// TwinCAT 3 PLC project MasterArmControl
// ProgramVersion: 3.1.4024.0
// libraries:
//   Tc2_Math, * (Beckhoff Automation GmbH)
//   Tc2_Standard, * (Beckhoff Automation GmbH)
//   Tc2_System, * (Beckhoff Automation GmbH)
//   Tc3_Module, * (Beckhoff Automation GmbH)
// project tree:
//   Controllers/ FB_ADD.TcPOU, FB_Test.TcPOU, ITF.TcIO
//   DUTs/Enum/ E_DriverCtrlWord.TcDUT, E_DriverOPMode.TcDUT (not stored), E_DriverStatusWord.TcDUT (not stored), E_InstrumentType.TcDUT, E_MasterArmState.TcDUT, E_MatchedSlaveArmIdx.TcDUT, E_SlaveArmState.TcDUT
//   DUTs/Structure/ ST_CartStatus.TcDUT, ST_Frame.TcDUT (not stored), ST_InstruStatus.TcDUT (not stored), ST_MasterStatus.TcDUT, ST_MotorInputs.TcDUT, ST_MotorOutputs.TcDUT (not stored), ST_SlaveStatus.TcDUT (not stored)
//   DUTs/Type/ Mat3d.TcDUT (not stored), Vec3d.TcDUT (not stored), Vec6d.TcDUT (not stored), Vec7d.TcDUT (not stored), Vec7i.TcDUT (not stored)
//   FBs_Controller/ FB_MasterArmCtrlBase.TcPOU, FB_PID.TcPOU (not stored), FBRedunOriControl.TcPOU, I_MasterArmCtrl.TcIO
//   FBs_dynamics/ FB_MasterGravity.TcPOU, FB_MasterGravity_1.TcPOU (not stored)
//   FBs_Filter/ FB_LowPassFilter.TcPOU (not stored)
//   GVLs/ GVL_ArmParameters.TcGVL, GVL_CartParameters.TcGVL, GVL_ControlParameters.TcGVL, GVL_MathDefine.TcGVL, GVL_MotorParameters.TcGVL (not stored), GVL_SafetyParameters.TcGVL (not stored), GVL_SystemParameters.TcGVL (not stored)
//   / MAIN.TcPOU, PlcTask.TcTTO (not stored)
//   Maths/ addVec3.TcPOU, atan2.TcPOU (not stored), cot.TcPOU, mat3Mat3.TcPOU (not stored), mat3Vec3.TcPOU, mat67Vec7.TcPOU, rotZ.TcPOU, rotY.TcPOU (not stored), rotX.TcPOU, transform.TcPOU
//   Robots/ FB_Joint.TcPOU, FB_MasterArm.TcPOU, FB_MasterRobot.TcPOU
// real-time tasks:
//   TASK PlcTask: cycle T#10ms, priority 20, ADS port 350

// ---- DUTs/Enum/E_DriverCtrlWord.TcDUT
TYPE E_DriverCtrlWord :
(
	DriverCtrlWord_INIT := 6,
	DriverCtrlWord_PREOP := 7,
	DriverCtrlWord_OP := 15
);
END_TYPE

// ---- DUTs/Enum/E_InstrumentType.TcDUT
TYPE E_InstrumentType :
(
	InstruType_UNKNOWM := 0,
	InstruType_endoscope := 1,
	InstruType_NeedleGripper := 2,
	InstruType_Energy :=3
);
END_TYPE

// ---- DUTs/Enum/E_MasterArmState.TcDUT
TYPE E_MasterArmState :
(
	MasterArmState_Errot := 0,
	MasterArmState_Cart := 1,
	MasterArmState_Init :=2,
	MasterArmState_Home :=3,
	MasterArmState_Standby :=4,
	MasterArmState_Matching :=5,
	MasterArmState_Ready :=6,
	MasterArmState_MasterSlave :=7,
	MasterArmState_Clutch :=8,
	MasterArmState_Endoscope :=9
);
END_TYPE

// ---- DUTs/Enum/E_MatchedSlaveArmIdx.TcDUT
TYPE E_MatchedSlaveArmIdx :
(
	MatchedSlaveArmIdx_NULL := 0,
	MatchedSlaveArmIdx_1 := 1,
	MatchedSlaveArmIdx_2 := 2,
	MatchedSlaveArmIdx_3 := 3,
	MatchedSlaveArmIdx_4 := 4
);
END_TYPE

// ---- DUTs/Enum/E_SlaveArmState.TcDUT
TYPE E_SlaveArmState :
(
	SlaveArmState_Errot := 0,
	SlaveArmState_Cart := 1,
	SlaveArmState_Init :=2,
	SlaveArmState_Standby :=3,
	SlaveArmState_InstallPanel:=4,
	SlaveArmState_PanelReady :=5,
	SlaveArmState_InstallInstru :=6,
	SlaveArmState_InstruReady :=7,
	SlaveArmState_MasterSlave :=8,
	SlaveArmState_InstallScope :=9,
	SlaveArmState_ScopeReady :=10,
	SlaveArmState_EndoScope :=11
);
END_TYPE

// ---- DUTs/Structure/ST_CartStatus.TcDUT
TYPE ST_CartStatus :
STRUCT
	m_monitorAngle:LREAL := 0.0;
	m_armSwitch:BOOL := FALSE;
	m_clutchSwitch:BOOL := FALSE;
	m_endoscopeSwitch:BOOL := FALSE;
	m_instrumentPowerSwitch:BOOL := FALSE;
	m_monitorAdjustSwitch:BOOL := FALSE;
	m_tableAdjustSwitch:BOOL := FALSE;
END_STRUCT
END_TYPE

// ---- DUTs/Structure/ST_MasterStatus.TcDUT
TYPE ST_MasterStatus :
STRUCT
	// state machine
	m_armState:ARRAY[1..g_mArmNum] OF E_masterArmState;
	
	// index(0 to 4) of slave arm which is tele-linked to master arm
	m_slaveArmIdx :ARRAY[1..g_mArmNum] OF INT;
	
	// grip angle
	m_gripAngle:ARRAY[1..g_mArmNum] OF LREAL;
	
	// command arm pose in monitor
	m_cmdArmPose :ARRAY[1..g_mArmNum] OF ST_Frame;
	
	// current arm pose in monitor
	m_curArmPose:ARRAY[1..g_mArmNum] OF ST_Frame;
	
	// command arm twist[linear velocity; angular veloicty] in monitor
	m_cmdArmTwist:ARRAY[1..g_mArmNum,1..6] OF LREAL;
	
	// current arm twist[linear velocity; angular veloicty] in monitor
	m_curArmTwist:ARRAY[1..g_mArmNum,1..6] OF LREAL;
	
	// joint position compute with motor encoder
	m_curMotorPos :ARRAY[1..g_mJntNum] OF LREAL;
	
	// joint position compute with link/abs encoder
	m_curLinkPos :ARRAY[1..g_mArmNum, 1..g_mJntNum] OF LREAL;
	
	// target joint position 
	m_cmdJntPos :ARRAY[1..g_mArmNum, 1..g_mJntNum] OF LREAL;
	
	// current joint position 
	m_curJntPos :ARRAY[1..g_mArmNum, 1..g_mJntNum] OF LREAL;
	
	// target joint velocity 
	m_cmdJntVel :ARRAY[1..g_mArmNum, 1..g_mJntNum] OF LREAL;
	
	// current joint position 
	m_curJntVel :ARRAY[1..g_mArmNum, 1..g_mJntNum] OF LREAL;
	
	// command joint torque 
	m_cmdJntTrq :ARRAY[1..g_mArmNum, 1..g_mJntNum] OF LREAL;
	
	// current joint torque 
	m_curJntTrq :ARRAY[1..g_mArmNum, 1..g_mJntNum] OF LREAL;
	
END_STRUCT
END_TYPE

// ---- DUTs/Structure/ST_MotorInputs.TcDUT
TYPE ST_MotorInputs:
STRUCT
	m_driverError:UDINT;
	m_statusWord:UINT;
	
	// motor/relative encoder from IO
	m_motorEncoder :DINT;
	
	// link/absolute encoder form IO
	m_linkEncoder :DINT;
	
	// motor current from IO
	m_current : DINT;
	
END_STRUCT
END_TYPE

// ---- GVLs/GVL_ArmParameters.TcGVL
// use slot attribute larger than 49990, which is the default one, if it depends on variable in other file
{attribute 'global_init_slot' := '49991'} 
VAR_GLOBAL CONSTANT 

// distance between shoulders of left and right arm
g_armShoulderDistance :LREAL := 0.5;
 	
(* 
% DH definetion
% !!!!NOTE: q4 is the DH joint position, NOT the motor one
% paramters definiton:
% d1: arm origin to joint1 
% a3: upper arm length
% a4: lower arm length
% d4: wrist height
% a9: parallel structure width
% DH definition:
% index     parent  alpha   a       theta   d       active
% 1         0       0       0       q1      d1      1
% 2         1       -90     0       q2      0       1
% 3         0       0       a3      q3      0       0
% 4         3       -90     a4      q4      d4      1
% 5         4       90      0       q5      0       1
% 6         5       -90     0       q6      0       1
% 7         6       90      0       q7      0       1

% 8         1       -90     0       q8      0       1
% 9         8       0       a9      q9      0       0
% 10        9       0       a3      q10     0       0
% 11        3       0       a9      0       0       fixed

%q4 = motor_q4+q8-q2-90
%q3 = q8 - q2;
%q9 = q2-q8;
%q10 = q8-q2

*)
	g_d1:LREAL:=0.26085;
	g_d4:LREAL:=0.1615;
	g_a3:LREAL:=0.278;
	g_a4:LREAL:=0.365;
	
	//alpha,a,d,theta	
	g_materArmDH:ARRAY[1..7,1..4] OF LREAL:=[0,		0,		g_d1,	0,      
											-pi/2,	0,		0,		0,
											0,		g_a3,	0,		0,
									        -pi/2,	g_a4,	g_d4,	0,       
											pi/2,	0,		0,		0,
								            -pi/2,	0,		0,		0,
							         		pi/2,	0,		0,		0];


// arm gravity parameters
(*graParam=[ 2.7244*m3 + 2.7244*m4 + 2.7244*m5 + 2.7244*m6 + 9.8*mx2 + 9.8*mx9,
			9.8*my2 + 9.8*my9,
			3.577*m4 + 3.577*m5 + 3.577*m6 + 0.49*m9 + 9.8*mx3 + 9.8*mx8
			1.5827*m4 + 1.5827*m5 + 1.5827*m6 + 9.8*my3 + 9.8*my8 + 9.8*mz4
			mz5-my4,	my5+mz6,  	mx4,   	mx5, 	mx6,   	my6
			preF2,   k2,   preF3,    k3,    preF5   k5]*)
g_gravityParam :ARRAY[1..2, 1..16] OF REAL := 
	[ 	4.22377, -0.000238508, 3.4348, 0.523733, -0.0377839, 0.0220708, 0.0000375, 0.0000351, 0.00001, -0.0147457, 
		12.4552, 2044.8, 12.4552, 2044.8, 2.13504, 403.2,
	 	3.95717, -0.000238508, 3.22352, 0.823427, -0.0371339, 0.0238336, 0.0000375, 0.0000117, -0.00001, -0.0145314, 
		13.7318, 1841.41, 12.4552, 2044.8, 2.13504, 403.2];
// spring parameters
// spring2 [L0, b1, b2, l1, r0]
g_spring2Param :ARRAY[1..5] OF LREAL :=[101.6E-3, 14.5E-3, 15E-3, 172E-3, 31E-3];
// spring3 [L0, b1, b2, l1, r0,d]
g_spring3Param :ARRAY[1..6] OF LREAL :=[101.6E-3, 14E-3, 15E-3, 172E-3, 30E-3, 10E-3];
// spring5 [L0, s1, L1, r0, beta]
g_spring5Param :ARRAY[1..5] OF LREAL :=[34.93E-3, 34.3E-3, 100E-3, 12.5E-3, 32.02*g_deg2rad];
END_VAR

// ---- GVLs/GVL_CartParameters.TcGVL
VAR_GLOBAL CONSTANT
	
	
	
	//car
(*	//tr_1:lreal:=deg2rad(0.556*0.001/360);  tr_2:lreal:=deg2rad(0.19*0.001/360);	
	line_enconder_car:ARRAY[1..4] OF DINT:=[line_1,line_1,line_1,line_1];
	transmission_ratio_car:ARRAY[1..4] OF LREAL:=[2*pi/0.0004682,3317.76,2*pi/0.0004682,1.5*138.0/5*2*pi/0.004];//2*pi/0.00014493];
	line_enconder_car_sec:ARRAY[1..4] OF DINT:=[line_2,line_2,line_2,line_2];
	transmission_ratio_car_sec:ARRAY[1..4] OF lreal:=[1,1,1,1];
	Line_Resolution_car:LREAL:=0.001*2/(EXPT(2,13));
	
	rad_12:LREAL:=deg2rad(12);  rad_80:LREAL:=deg2rad(80);  	rad_20:LREAL:=deg2rad(20);   rad_7:LREAL:=deg2rad(7); 
	rad_31:LREAL:=deg2rad(31.6483);rad_2:LREAL:=deg2rad(2.6183);
	//vel_max_car:ARRAY[1..4] OF LREAL:=[0.048,rad_12,0.032,0.025];
	vel_max_car:ARRAY[1..4] OF LREAL:=[0.048*0.3,rad_12*0.2,0.032*0.3,0.025*0.3];
	
	//acc_max_car:ARRAY[1..4] OF LREAL:=[0.3,rad_80,0.2,0.15];
	acc_max_car:ARRAY[1..4] OF LREAL:=[0.048*2,rad_12*2,0.032*2,0.025*2];
	//***MODIFY-2022***旋转监视器极限位置修改
	distance_min_car:ARRAY[1..4] OF LREAL:=[0,-rad_31,0,0];//[0.0065,-rad_73,0.029,0.004];
	distance_max_car:ARRAY[1..4] OF LREAL:=[0.38,rad_2,0.240,0.20];//[0.3565,0,0.164,0.184];
	
	torque_constant_car:ARRAY[1..4] OF lreal:=[0.0292,0.0292,0.0292,0.0292];
	torque_max_car:ARRAY[1..4] OF lreal:=[1000,1000,1000,1000];
	//current_peak_car:ARRAY[1..4] OF LREAL:=[41200,41200,41200,41200];
	current_peak_car:ARRAY[1..4] OF LREAL:=[3800*2,3800*2,3800*2,3800*2];
	
	transmition_efficiency_car:ARRAY[1..4] OF LREAL:=[0.69,0.28,0.69,0.24];
	current_related_car:ARRAY[1..4] OF lreal:=[3800,3800,3800,3800];
	
	Car_relative_encoder_Offset:ARRAY[1..4] OF lreal;	
	Car_Motion_direction:ARRAY[1..4] OF lreal;
	Car_Absolute_encoder_direction:ARRAY[1..4] OF LREAL;
	
	length_second_encoder_resolution_car:ARRAY[1..4] OF LREAL:=[Line_Resolution_car,6.71/16777216,Line_Resolution_car,Line_Resolution_car];	
	//length_second_encoder_car:ARRAY[1..4] OF LREAL:=[6.71,6.71,6.71,6.71];	
	Car_Target_position_error:ARRAY[1..4] OF LREAL:=[0.001,1.0/57,0.001,0.001];*)
END_VAR

// ---- GVLs/GVL_ControlParameters.TcGVL
VAR_GLOBAL CONSTANT
	// master arm joint position controller parameters
	g_posKp :ARRAY[1..7] OF LREAL :=[0.0, 0.0, 0.0, 0.0, 0.0, 0.0, 0.0];
	g_posKd :ARRAY[1..7] OF LREAL :=[0.0, 0.0, 0.0, 0.0, 0.0, 0.0, 0.0];
	g_posKi :ARRAY[1..7] OF LREAL :=[0.0, 0.0, 0.0, 0.0, 0.0, 0.0, 0.0];
	g_posKiLimit :ARRAY[1..7] OF LREAL :=[500,500,500,500,100,100,100];// define in current
	g_posCtrlLimit :ARRAY[1..7] OF LREAL :=[1000,1000,1000,1000,200,200,200];// define in current
	
	// filter cut-off frequency for velocity and torque
	g_curJntVelLpfCutoffFreq :LREAL := 30;
	g_cmdJntPosLpfCutoffFreq :LREAL := 30;
	g_cmdJntTrqLpfCutoffFreq :LREAL := 300;
	
END_VAR

// ---- GVLs/GVL_MathDefine.TcGVL
VAR_GLOBAL CONSTANT
	g_smallNum :LREAL := 1E-8;
	g_deg2Rad :LREAL := pi/180.0;
	g_rad2Deg :LREAL := 180.0/pi;
	g_eye3d :Mat3d:=[1, 0, 0,
					 0, 1, 0,
					 0, 0, 1];
	g_zeorMat3d :Mat3d:=[9(0)];
	g_zeroVec3d :Vec3d:= [3(0)];
	
END_VAR

// ---- Controllers/ITF.TcIO
INTERFACE ITF

END_INTERFACE

// ---- FBs_Controller/I_MasterArmCtrl.TcIO
INTERFACE I_MasterArmCtrl

METHOD reset : BOOL
VAR_INPUT
END_VAR
END_METHOD

METHOD run : BOOL
VAR_IN_OUT CONSTANT
	i_shoulderPose :ARRAY[1..2] OF ST_Frame;
	i_slaveStatus :ST_SlaveStatus;
END_VAR
VAR_IN_OUT
	i_masterArms :ARRAY[1..g_mArmNum] OF FB_MasterArm;
END_VAR
END_METHOD

END_INTERFACE

// ---- Controllers/FB_ADD.TcPOU
FUNCTION_BLOCK PUBLIC FB_ADD
VAR_INPUT
END_VAR
VAR_OUTPUT
END_VAR
VAR
END_VAR

END_FUNCTION_BLOCK

// ---- Controllers/FB_Test.TcPOU
FUNCTION_BLOCK FB_Test
VAR_INPUT
END_VAR
VAR_OUTPUT
END_VAR
VAR
END_VAR

END_FUNCTION_BLOCK

// ---- FBs_Controller/FB_MasterArmCtrlBase.TcPOU
FUNCTION_BLOCK FB_MasterArmCtrlBase IMPLEMENTS I_MasterArmCtrl
VAR_INPUT
END_VAR
VAR_OUTPUT
END_VAR
VAR
	// flag if enter controller for the first time
	m_firstIn:BOOL:=TRUE;
	
	// arm control data
	m_cmdJntPos :ARRAY[1..g_mArmNum] OF VEC7d;
	m_cmdJntVel :ARRAY[1..g_mArmNum] OF VEC7d;
	m_cmdJntTrq :ARRAY[1..g_mArmNum] OF VEC7d;
	m_jntOPMode :ARRAY[1..g_mArmNum] OF Vec7i;
END_VAR

// override this function in each exact controller
METHOD PROTECTED calcCmdJntPos : BOOL
VAR_IN_OUT CONSTANT
	i_shoulderPose :ARRAY[1..2] OF ST_Frame;
	i_slaveStatus :ST_SlaveStatus;
END_VAR
VAR_IN_OUT
	i_masterArms :ARRAY[1..g_mArmNum] OF FB_MasterArm;
END_VAR
END_METHOD

// override this function in each exact controller
METHOD PROTECTED calcCmdJntTrq : BOOL
VAR_IN_OUT CONSTANT
	i_shoulderPose :ARRAY[1..2] OF ST_Frame;
	i_slaveStatus :ST_SlaveStatus;
END_VAR
VAR_IN_OUT
	i_masterArms :ARRAY[1..g_mArmNum] OF FB_MasterArm;
END_VAR
END_METHOD

// override this function in each exact controller
// NOTICE: set joint control mode here, and do some initialization if needed
METHOD PROTECTED Init : BOOL
VAR_IN_OUT CONSTANT
	i_masterArms	: ARRAY [1..g_mArmNum] OF FB_MasterArm;
END_VAR
VAR
	i,j:INT;
END_VAR
FOR i:=1 TO g_mArmNum DO
	m_cmdJntPos[i]:=i_masterArms[i].curJntPos;
	FOR j:=1 TO g_mJntNum DO
		m_cmdJntVel[i][j]:=0.0;
		m_cmdJntTrq[i][j]:=0.0;
		m_jntOPMode[i][j]:=DriverOPMode_Pos;
	END_FOR
END_FOR
END_METHOD

{warning '添加方法实现'}
METHOD reset : BOOL
m_firstIn:=true;
END_METHOD

{warning '添加方法实现'}
METHOD run : BOOL
VAR_IN_OUT CONSTANT
	i_shoulderPose :ARRAY[1..2] OF ST_Frame;
	i_slaveStatus :ST_SlaveStatus;
END_VAR
VAR_IN_OUT
	i_masterArms :ARRAY[1..g_mArmNum] OF FB_MasterArm;
END_VAR

VAR
	i:INT;
END_VAR
IF m_firstIn THEN
	Init(i_masterArms);
	m_firstIn:=FALSE;
END_IF

// calculate command joint position
calcCmdJntPos(i_shoulderPose,i_slaveStatus,i_masterArms);

// calculate command joint torque
calcCmdJntTrq(i_shoulderPose,i_slaveStatus,i_masterArms);

// update commands to arm
FOR i:=1 TO g_mArmNum DO
	i_masterArms[i].cmdJntPos:=m_cmdJntPos[i];
	i_masterArms[i].cmdJntVel:=m_cmdJntVel[i];
	i_masterArms[i].cmdJntTrq:=m_cmdJntTrq[i];
	i_masterArms[i].jntOPMode:=m_jntOPMode[i];
END_FOR
END_METHOD

END_FUNCTION_BLOCK

// ---- Robots/FB_MasterArm.TcPOU
FUNCTION_BLOCK FB_MasterArm
// NOTICE: all joints are the ture active joints, not DH ones!
VAR_INPUT
END_VAR
VAR_OUTPUT
END_VAR
VAR
	// arm index, 0 for left arm, 1 for right arm
	m_armIdx: INT;
	
	// grip angle from hall sensor IO
	m_gripHallSensorValue AT%I* :UDINT;
	m_gripAngle :LREAL;
	
	// arm block
	m_joints :ARRAY[1..g_mJntNum] OF FB_Joint;
	
	// arm cartesian data, defined in each arm origin
	m_curCartPose	:ST_Frame;
	m_curCartTwist:ARRAY[1..g_cartDofs] OF LREAL;
	
	// arm joint data
	m_curJntPos :Vec7d;
	m_curJntVel :Vec7d;
	m_curJntTrq :Vec7d;
	m_cmdJntPos :Vec7d;
	m_cmdJntVel :Vec7d;
	m_cmdJntTrq :Vec7d;
	m_jntOPMode :Vec7i;
	
	// arm daynamic data
	m_jntGravity :ARRAY[1..g_mJntNum] OF LREAL;
	
	// arm jacobian 
	m_jaco :ARRAY[1..g_cartDofs, 1..g_mJntNum] OF LREAL;
	
	// joint position controller
	m_jntPIDCtrl :ARRAY[1..g_mJntNum] OF FB_PID;
	
	// grivity model
	m_gravityModel : FB_MasterGravity;
	
END_VAR

// TODO
METHOD PROTECTED calcGripAngle : LREAL
VAR_INPUT
END_VAR
END_METHOD

METHOD PUBLIC calcJaco : BOOL
VAR_IN_OUT CONSTANT
	i_jntPos :ARRAY[1..g_mJntNum] OF LREAL;
END_VAR
VAR_IN_OUT
	r_jaco :ARRAY[1..g_cartDofs, 1..g_mJntNum] OF LREAL;
END_VAR
VAR_INPUT
END_VAR

VAR
	q1,q2, q3, q4, q5, q6, q7 :LREAL;
	d1,d4,a3,a4 :LREAL;
	j:INT;
END_VAR
// !Convert active joint position to DH model for kinematic calculation
q1:=i_jntPos[1];  
q2:=i_jntPos[2];  
q3:=i_jntPos[3]-i_jntPos[2];  //q3=q8-q2
q4:=i_jntPos[4]+i_jntPos[3]-i_jntPos[2]-pi/2;//q4DH=q4motor+q8-q2-90;  
q5:=i_jntPos[5];  
q6:=i_jntPos[6];  
q7:=i_jntPos[7];  
d1:=g_d1;
d4:=g_d4;
a3:=g_a3;
a4:=g_a4;

// jacobian with DH joints
r_jaco[1,1]:=-SIN(q1)*(COS(q2)*(a3 + a4*COS(q3) - d4*SIN(q3)) - SIN(q2)*(d4*COS(q3) + a4*SIN(q3))) ;
r_jaco[1,2]:=-COS(q1)*(SIN(q2)*(a3 + a4*COS(q3) - d4*SIN(q3)) + COS(q2)*(d4*COS(q3) + a4*SIN(q3))) ;
r_jaco[1,3]:=-COS(q1)*(d4*COS(q2 + q3) + a4*SIN(q2 + q3)) ;
r_jaco[1,4]:=0 ;
r_jaco[1,5]:=0 ;
r_jaco[1,6]:=0 ;
r_jaco[1,7]:=0;
 
r_jaco[2,1]:=COS(q1)*(COS(q2)*(a3 + a4*COS(q3) - d4*SIN(q3)) - SIN(q2)*(d4*COS(q3) + a4*SIN(q3))); 
r_jaco[2,2]:=-SIN(q1)*(SIN(q2)*(a3 + a4*COS(q3) - d4*SIN(q3)) + COS(q2)*(d4*COS(q3) + a4*SIN(q3))); 
r_jaco[2,3]:=-SIN(q1)*(d4*COS(q2 + q3) + a4*SIN(q2 + q3)); 
r_jaco[2,4]:=0; 
r_jaco[2,5]:=0; 
r_jaco[2,6]:=0; 
r_jaco[2,7]:=0;

 
r_jaco[3,1]:=0 ;
r_jaco[3,2]:=- COS(q1)*(COS(q1)*COS(q2)*(a3 + a4*COS(q3) - d4*SIN(q3)) - COS(q1)*SIN(q2)*(d4*COS(q3) + a4*SIN(q3))) - SIN(q1)*(COS(q2)*SIN(q1)*(a3 + a4*COS(q3) - d4*SIN(q3)) - SIN(q1)*SIN(q2)*(d4*COS(q3) + a4*SIN(q3)));
r_jaco[3,3]:=- COS(q1)*(a4*COS(q2 + q3)*COS(q1) - d4*SIN(q2 + q3)*COS(q1)) - SIN(q1)*(a4*COS(q2 + q3)*SIN(q1) - d4*SIN(q2 + q3)*SIN(q1));
r_jaco[3,4]:=0;
r_jaco[3,5]:=0;
r_jaco[3,6]:=0 ;
r_jaco[3,7]:=0 ;

r_jaco[4,1]:=0 ;
r_jaco[4,2]:=-SIN(q1) ;
r_jaco[4,3]:=-SIN(q1) ;
r_jaco[4,4]:=-SIN(q2 + q3)*COS(q1) ;
r_jaco[4,5]:=COS(q2 + q3)*COS(q1)*SIN(q4) - COS(q4)*SIN(q1) ;
r_jaco[4,6]:=- SIN(q5)*(SIN(q1)*SIN(q4) + COS(q2 + q3)*COS(q1)*COS(q4)) - SIN(q2 + q3)*COS(q1)*COS(q5) ;
r_jaco[4,7]:=SIN(q6)*(COS(q5)*(SIN(q1)*SIN(q4) + COS(q4)*(COS(q1)*COS(q2)*COS(q3) - COS(q1)*SIN(q2)*SIN(q3))) - SIN(q5)*(COS(q1)*COS(q2)*SIN(q3) + COS(q1)*COS(q3)*SIN(q2))) - COS(q6)*(COS(q4)*SIN(q1) - SIN(q4)*(COS(q1)*COS(q2)*COS(q3) - COS(q1)*SIN(q2)*SIN(q3)));
 
r_jaco[5,1]:=0; 
r_jaco[5,2]:=COS(q1); 
r_jaco[5,3]:=COS(q1); 
r_jaco[5,4]:=-SIN(q2 + q3)*SIN(q1); 
r_jaco[5,5]:=COS(q1)*COS(q4) + COS(q2 + q3)*SIN(q1)*SIN(q4); 
r_jaco[5,6]:=SIN(q5)*(COS(q1)*SIN(q4) - COS(q2 + q3)*COS(q4)*SIN(q1)) - SIN(q2 + q3)*COS(q5)*SIN(q1); 
r_jaco[5,7]:=COS(q6)*(COS(q1)*COS(q4) - SIN(q4)*(SIN(q1)*SIN(q2)*SIN(q3) - COS(q2)*COS(q3)*SIN(q1))) - SIN(q6)*(COS(q5)*(COS(q1)*SIN(q4) + COS(q4)*(SIN(q1)*SIN(q2)*SIN(q3) - COS(q2)*COS(q3)*SIN(q1))) + SIN(q5)*(COS(q2)*SIN(q1)*SIN(q3) + COS(q3)*SIN(q1)*SIN(q2)));

r_jaco[6,1]:=1 ;
r_jaco[6,2]:=0 ;
r_jaco[6,3]:=0 ;
r_jaco[6,4]:=-COS(q2 + q3) ;
r_jaco[6,5]:=-SIN(q2 + q3)*SIN(q4) ;
r_jaco[6,6]:=SIN(q2 + q3)*COS(q4)*SIN(q5) - COS(q2 + q3)*COS(q5) ;
r_jaco[6,7]:=- SIN(q6)*(COS(q2 + q3)*SIN(q5) + SIN(q2 + q3)*COS(q4)*COS(q5)) - SIN(q2 + q3)*COS(q6)*SIN(q4);

// jacobian with active joints
// jaco_DH*qdot_DH = jaco_DH * (A * qdot)= jaco * qdot
// A =[ 1  0 0 0 0 0 0
//		0  1 0 0 0 0 0
//		0 -1 1 0 0 0 0
//		0 -1 1 1 0 0 0
//		0 0  0 0 1 0 0
//      0 0  0 0 0 1 0
// 		0 0  0 0 0 0 1]
 FOR j:=1 TO 6 DO 
	 r_jaco[j,2]:=r_jaco[j,2]-r_jaco[j,3]-r_jaco[j,4];
	 r_jaco[j,3]:=r_jaco[j,3]+r_jaco[j,4];
 END_FOR
END_METHOD

PROPERTY cmdJntPos : Vec7d
GET
cmdJntPos:=m_cmdJntPos;
END_GET
SET
m_cmdJntPos:=cmdJntPos;
END_SET
END_PROPERTY

PROPERTY cmdJntTrq : Vec7d
GET
cmdJntTrq:=m_cmdJntTrq;
END_GET
SET
m_cmdJntTrq:=cmdJntTrq;
END_SET
END_PROPERTY

PROPERTY cmdJntVel : Vec7d
GET
cmdJntVel :=m_cmdJntVel;
END_GET
SET
m_cmdJntVel :=cmdJntVel;
END_SET
END_PROPERTY

PROPERTY curCartPose : ST_Frame
GET
curCartPose :=m_curCartPose;
END_GET
END_PROPERTY

PROPERTY curCartTwist : Vec6d
GET
curCartTwist :=m_curCartTwist;
END_GET
END_PROPERTY

PROPERTY curJntPos : Vec7d
GET
curJntPos:=m_curJntPos;
END_GET
SET
m_curJntPos:=curJntPos;
END_SET
END_PROPERTY

PROPERTY curJntTrq : Vec7d
GET
curJntTrq:=m_curJntTrq;
END_GET
SET
m_curJntTrq:=curJntTrq;
END_SET
END_PROPERTY

PROPERTY curJntVel : Vec7d
GET
curJntVel:=m_curJntVel;
END_GET
SET
m_curJntVel:=curJntVel;
END_SET
END_PROPERTY

METHOD PUBLIC diable : BOOL
VAR_IN_OUT CONSTANT
	i_jntIdx :Vec7i;
END_VAR
VAR
	i :INT ;
END_VAR
FOR i:=1 TO g_mJntNum DO
	IF 1= i_jntIdx[i] THEN
		m_joints[i].disable();
	END_IF
END_FOR
END_METHOD

METHOD PUBLIC enable : BOOL
VAR_IN_OUT CONSTANT
	i_jntIdx :Vec7i;
END_VAR
VAR
	i :INT ;
END_VAR
enable := TRUE;
FOR i:=1 TO g_mJntNum DO
	IF 1= i_jntIdx[i] THEN
		enable := enable AND m_joints[i].enable();
	END_IF
END_FOR
END_METHOD

// from active joint position to cartesian pose in arm origin
METHOD PROTECTED forwardKinematic : BOOL
VAR_IN_OUT CONSTANT
	i_jntPos :ARRAY[1..g_mJntNum] OF LREAL;
END_VAR
VAR_IN_OUT
	r_curCartPose :ST_Frame;
END_VAR
VAR
	q1,q2, q3, q4, q5, q6, q7 :LREAL;
	d1,d4,a3,a4 :LREAL;
END_VAR
// !Convert active joint position to DH model for kinematic calculation
q1:=i_jntPos[1];  
q2:=i_jntPos[2];  
q3:=i_jntPos[3]-i_jntPos[2];  //q3=q8-q2
q4:=i_jntPos[4]+i_jntPos[3]-i_jntPos[2]-pi/2;//q4DH=q4motor+q8-q2-90;  
q5:=i_jntPos[5];  
q6:=i_jntPos[6];  
q7:=i_jntPos[7];  
d1:=g_d1;
d4:=g_d4;
a3:=g_a3;
a4:=g_a4;

// cartesian pose frame
r_curCartPose.m_pos[1]:=COS(q1)*(a4*COS(q2 + q3) - d4*SIN(q2 + q3) + a3*COS(q2)); 
r_curCartPose.m_pos[2]:=SIN(q1)*(a4*COS(q2 + q3) - d4*SIN(q2 + q3) + a3*COS(q2)); 
r_curCartPose.m_pos[3]:=d1 - d4*COS(q2 + q3) - a4*SIN(q2 + q3) - a3*SIN(q2); 
r_curCartPose.m_rot[1,1]:=COS(q7)*(SIN(q6)*(COS(q4)*SIN(q1) - SIN(q4)*(COS(q1)*COS(q2)*COS(q3) - COS(q1)*SIN(q2)*SIN(q3))) + COS(q6)*(COS(q5)*(SIN(q1)*SIN(q4) + COS(q4)*(COS(q1)*COS(q2)*COS(q3) - COS(q1)*SIN(q2)*SIN(q3))) - SIN(q5)*(COS(q1)*COS(q2)*SIN(q3) + COS(q1)*COS(q3)*SIN(q2)))) - SIN(q7)*(SIN(q5)*(SIN(q1)*SIN(q4) + COS(q4)*(COS(q1)*COS(q2)*COS(q3) - COS(q1)*SIN(q2)*SIN(q3))) + COS(q5)*(COS(q1)*COS(q2)*SIN(q3) + COS(q1)*COS(q3)*SIN(q2)));
r_curCartPose.m_rot[2,1]:=SIN(q7)*(SIN(q5)*(COS(q1)*SIN(q4) + COS(q4)*(SIN(q1)*SIN(q2)*SIN(q3) - COS(q2)*COS(q3)*SIN(q1))) - COS(q5)*(COS(q2)*SIN(q1)*SIN(q3) + COS(q3)*SIN(q1)*SIN(q2))) - COS(q7)*(SIN(q6)*(COS(q1)*COS(q4) - SIN(q4)*(SIN(q1)*SIN(q2)*SIN(q3) - COS(q2)*COS(q3)*SIN(q1))) + COS(q6)*(COS(q5)*(COS(q1)*SIN(q4) + COS(q4)*(SIN(q1)*SIN(q2)*SIN(q3) - COS(q2)*COS(q3)*SIN(q1))) + SIN(q5)*(COS(q2)*SIN(q1)*SIN(q3) + COS(q3)*SIN(q1)*SIN(q2))));
r_curCartPose.m_rot[3,1]:=- SIN(q7)*(COS(q2 + q3)*COS(q5) - SIN(q2 + q3)*COS(q4)*SIN(q5)) - COS(q7)*(COS(q2 + q3)*COS(q6)*SIN(q5) - SIN(q2 + q3)*SIN(q4)*SIN(q6) + SIN(q2 + q3)*COS(q4)*COS(q5)*COS(q6)); 
r_curCartPose.m_rot[1,2]:=- SIN(q7)*(SIN(q6)*(COS(q4)*SIN(q1) - SIN(q4)*(COS(q1)*COS(q2)*COS(q3) - COS(q1)*SIN(q2)*SIN(q3))) + COS(q6)*(COS(q5)*(SIN(q1)*SIN(q4) + COS(q4)*(COS(q1)*COS(q2)*COS(q3) - COS(q1)*SIN(q2)*SIN(q3))) - SIN(q5)*(COS(q1)*COS(q2)*SIN(q3) + COS(q1)*COS(q3)*SIN(q2)))) - COS(q7)*(SIN(q5)*(SIN(q1)*SIN(q4) + COS(q4)*(COS(q1)*COS(q2)*COS(q3) - COS(q1)*SIN(q2)*SIN(q3))) + COS(q5)*(COS(q1)*COS(q2)*SIN(q3) + COS(q1)*COS(q3)*SIN(q2))); 
r_curCartPose.m_rot[2,2]:=SIN(q7)*(SIN(q6)*(COS(q1)*COS(q4) - SIN(q4)*(SIN(q1)*SIN(q2)*SIN(q3) - COS(q2)*COS(q3)*SIN(q1))) + COS(q6)*(COS(q5)*(COS(q1)*SIN(q4) + COS(q4)*(SIN(q1)*SIN(q2)*SIN(q3) - COS(q2)*COS(q3)*SIN(q1))) + SIN(q5)*(COS(q2)*SIN(q1)*SIN(q3) + COS(q3)*SIN(q1)*SIN(q2)))) + COS(q7)*(SIN(q5)*(COS(q1)*SIN(q4) + COS(q4)*(SIN(q1)*SIN(q2)*SIN(q3) - COS(q2)*COS(q3)*SIN(q1))) - COS(q5)*(COS(q2)*SIN(q1)*SIN(q3) + COS(q3)*SIN(q1)*SIN(q2))); 
r_curCartPose.m_rot[3,2]:=SIN(q7)*(COS(q2 + q3)*COS(q6)*SIN(q5) - SIN(q2 + q3)*SIN(q4)*SIN(q6) + SIN(q2 + q3)*COS(q4)*COS(q5)*COS(q6)) - COS(q7)*(COS(q2 + q3)*COS(q5) - SIN(q2 + q3)*COS(q4)*SIN(q5)); 
r_curCartPose.m_rot[1,3]:=SIN(q6)*(COS(q5)*(SIN(q1)*SIN(q4) + COS(q4)*(COS(q1)*COS(q2)*COS(q3) - COS(q1)*SIN(q2)*SIN(q3))) - SIN(q5)*(COS(q1)*COS(q2)*SIN(q3) + COS(q1)*COS(q3)*SIN(q2))) - COS(q6)*(COS(q4)*SIN(q1) - SIN(q4)*(COS(q1)*COS(q2)*COS(q3) - COS(q1)*SIN(q2)*SIN(q3))); 
r_curCartPose.m_rot[2,3]:=COS(q6)*(COS(q1)*COS(q4) - SIN(q4)*(SIN(q1)*SIN(q2)*SIN(q3) - COS(q2)*COS(q3)*SIN(q1))) - SIN(q6)*(COS(q5)*(COS(q1)*SIN(q4) + COS(q4)*(SIN(q1)*SIN(q2)*SIN(q3) - COS(q2)*COS(q3)*SIN(q1))) + SIN(q5)*(COS(q2)*SIN(q1)*SIN(q3) + COS(q3)*SIN(q1)*SIN(q2)));
r_curCartPose.m_rot[3,3]:=- SIN(q6)*(COS(q2 + q3)*SIN(q5) + SIN(q2 + q3)*COS(q4)*COS(q5)) - SIN(q2 + q3)*COS(q6)*SIN(q4);
END_METHOD

PROPERTY gripAngle : LREAL
GET
gripAngle:=m_gripAngle;
END_GET
END_PROPERTY

METHOD PUBLIC init : BOOL
VAR_INPUT
	i_armIdx:INT;
END_VAR
VAR 
	i :INT ;
	currentRatioMotor2Jnt: LREAL;
END_VAR
m_armIdx:=i_armIdx;
m_gripAngle:=0;

FOR i:=1 TO g_mJntNum DO
	m_joints[i].init(m_armIdx, i);
END_FOR

m_gravityModel.init(m_armIdx);

// get joint data
FOR i:=1 TO g_mJntNum DO
	m_curJntPos[i] := m_joints[i].jntPos;
	m_curJntVel[i] := m_joints[i].jntVel;
	m_curJntTrq[i] := m_joints[i].jntTrq;
	m_cmdJntPos[i] := m_curJntPos[i];
	m_cmdJntVel[i] := 0.0;
	m_cmdJntTrq[i] := 0.0;
	m_jntOPMode[i] := DriverOPMode_Pos;
END_FOR 

// compute cartesion pose
forwardKinematic(i_jntPos:=m_curJntPos,r_curCartPose:=m_curCartPose);
FOR i:=1 TO g_cartDofs DO
	m_curCartTwist[i]:=0;
END_FOR

// compute jacobian
calcJaco(i_jntPos:=m_curJntPos,r_jaco:=m_jaco);

// joint controller init
FOR i:=1 TO g_mJntNum DO 
	currentRatioMotor2Jnt:=g_motorTrqConst[i]*g_motorReduction[i]/1000;
	m_jntPIDCtrl[i].init(g_armControlLoopInterval,g_posKp[i],g_posKd[i],g_posKi[i],
		g_posKiLimit[i]* currentRatioMotor2Jnt,	g_posCtrlLimit[i]*currentRatioMotor2Jnt);
END_FOR
END_METHOD

// from cartesian pose in arm origin to active joint position
METHOD PUBLIC inverseKinematic : BOOL
VAR_INPUT
	q4:LREAL;
	solution_ID:INT;
END_VAR
VAR_IN_OUT CONSTANT
	i_curCartPose :ST_Frame;
END_VAR
VAR_IN_OUT
	r_jntPos :ARRAY[1..g_mJntNum] OF LREAL;
END_VAR
VAR
	a3,a4,d1,d4:LREAL;
	px,py,pz:lreal;
	nx,ny,nz:lreal;
	ox,oy,oz:lreal;
	ax,ay,az:lreal;

	q1,q2,q3,q5,q6,q7:LREAL;
	
	q11,q12:LREAL;
	k1,A,B,C,fi,R0,q21,q22:lreal;
	ins1,ins2:lreal;
	
	A11,A12,A21,A22,C1,C2:lreal;
	SIN23,COS23,q23:lreal;
	
	T_74_left_23,q61,q62:lreal;
	T_74_left_13,T_74_left_33:lreal;
	T_74_left_21,T_74_left_22:LREAL;	
	
	succeed_1,succeed_2,succeed:BOOL;
END_VAR


//***********************单臂逆向运动学**************************//
d1:=g_d1;
d4:=g_d4;
a3:=g_a3;
a4:=g_a4;

nx:=i_curCartPose.m_rot[1,1];  ny:=i_curCartPose.m_rot[2,1];  nz:=i_curCartPose.m_rot[3,1];
ox:=i_curCartPose.m_rot[1,2]; oy:=i_curCartPose.m_rot[2,2];  oz:=i_curCartPose.m_rot[3,2];
ax:=i_curCartPose.m_rot[1,3];  ay:=i_curCartPose.m_rot[2,3];  az:=i_curCartPose.m_rot[3,3];
px:=i_curCartPose.m_pos[1]; py:=i_curCartPose.m_pos[2]; pz:=i_curCartPose.m_pos[3];


//求解q1
q11:=atan2(y:= py, x:= px);
q12:=-q11;
IF (Solution_ID<=4) THEN
	q1:=q11;
ELSE
	q1:=q12;
END_IF



//求解q2
k1:=px*COS(q1) + py*SIN(q1);
A:=2*a3*pz - 2*a3*d1;
B:=2*a3*k1;
C:=a3*a3 - a4*a4 + d1*d1 - 2*d1*pz - d4*d4 + k1*k1 + pz*pz;
fi:=atan2(y:= B, x:= A);

R0:=SQRT(A*A+B*B);

//*************程序保护性处理，避免软件崩溃***************//
IF ABS(C/R0)>1 THEN
	succeed_1:=FALSE;
	succeed:=FALSE;
	RETURN;
ELSE
	succeed_1:=TRUE;
END_IF

ins1:=atan2(y:= C/R0, x:= SQRT(1-(C/R0)*(C/R0)));
q21:=fi-ins1;
ins2:=atan2(y:= C/R0, x:= -SQRT(1-(C/R0)*(C/R0)));
q22:=fi-ins2;

IF (Solution_ID=1) OR (Solution_ID=2) OR (Solution_ID=5) OR (Solution_ID=6) THEN
	q2:=q21;
ELSE
	q2:=q22;
END_IF




//求解q3
A11:=- d4;
A12:=a4;
A21:=- a4;
A22:=-d4;
C1:=k1- a3*COS(q2);
C2:=pz - d1 + a3*SIN(q2);
sin23:=(C1*A22-C2*A12)/(A11*A22-A21*A12);
cos23:=(C2*A11-C1*A21)/(A11*A22-A21*A12);
q23:=atan2(y:= sin23, x:= cos23);
q3:=q23-q2;




//求解q6
T_74_left_23:=ax*(COS(q4)*SIN(q1) - COS(q1)*COS(q2)*COS(q3)*SIN(q4) + COS(q1)*SIN(q2)*SIN(q3)*SIN(q4)) - ay*(COS(q1)*COS(q4) + COS(q2)*COS(q3)*SIN(q1)*SIN(q4) - SIN(q1)*SIN(q2)*SIN(q3)*SIN(q4)) + az*SIN(q2 + q3)*SIN(q4);

//*************程序保护性处理，避免软件崩溃***************//
IF ABS(T_74_left_23>1) THEN
	succeed_2:=FALSE;
	succeed:=FALSE;
	RETURN;
ELSE
	succeed_2:=TRUE;
END_IF

q61:=ACOS(-T_74_left_23);
q62:=-ACOS(-T_74_left_23);
IF (Solution_ID=1) OR (Solution_ID=3) OR (Solution_ID=5) OR (Solution_ID=7) THEN
	q6:=q61;
ELSE
	q6:=q62;
END_IF


//求解q5
T_74_left_13:=ax*(SIN(q1)*SIN(q4) + COS(q1)*COS(q2)*COS(q3)*COS(q4) - COS(q1)*COS(q4)*SIN(q2)*SIN(q3)) - ay*(COS(q1)*SIN(q4) - COS(q2)*COS(q3)*COS(q4)*SIN(q1) + COS(q4)*SIN(q1)*SIN(q2)*SIN(q3)) - az*SIN(q2 + q3)*COS(q4);
T_74_left_33:=- az*COS(q2 + q3) - ax*SIN(q2 + q3)*COS(q1) - ay*SIN(q2 + q3)*SIN(q1);
q5:=atan2(y:= T_74_left_33*SIN(q6), x:= T_74_left_13*SIN(q6));


//求解q7
T_74_left_21:=nx*(COS(q4)*SIN(q1) - COS(q1)*COS(q2)*COS(q3)*SIN(q4) + COS(q1)*SIN(q2)*SIN(q3)*SIN(q4)) - ny*(COS(q1)*COS(q4) + COS(q2)*COS(q3)*SIN(q1)*SIN(q4) - SIN(q1)*SIN(q2)*SIN(q3)*SIN(q4)) + nz*SIN(q2 + q3)*SIN(q4);
T_74_left_22:=ox*(COS(q4)*SIN(q1) - COS(q1)*COS(q2)*COS(q3)*SIN(q4) + COS(q1)*SIN(q2)*SIN(q3)*SIN(q4)) - oy*(COS(q1)*COS(q4) + COS(q2)*COS(q3)*SIN(q1)*SIN(q4) - SIN(q1)*SIN(q2)*SIN(q3)*SIN(q4)) + oz*SIN(q2 + q3)*SIN(q4);
q7:=atan2(y:= -T_74_left_22*SIN(q6), x:= T_74_left_21*SIN(q6));


//! convert DH joint postion to active joint position
r_jntPos[1]:=q1;
r_jntPos[2]:=q2;
r_jntPos[3]:=q3+q2; // q8 = q3+q2
r_jntPos[4]:=q4+q2-r_jntPos[3]+pi/2;//q4DH=q4motor+q8-q2-90;  
r_jntPos[5]:=q5;
r_jntPos[6]:=q6;
r_jntPos[7]:=q7;

succeed:=TRUE;
inverseKinematic:=succeed;
END_METHOD

PROPERTY jntGravity : Vec7d
GET
jntGravity:=m_jntGravity;
END_GET
SET
m_jntGravity:=jntGravity;
END_SET
END_PROPERTY

PROPERTY jntOPMode : Vec7i
GET
jntOPMode:=m_jntOPMode;
END_GET
SET
m_jntOPMode:=jntOPMode;
END_SET
END_PROPERTY

// update joints control command
METHOD PUBLIC updateCmds : BOOL
VAR_INPUT
END_VAR
VAR
	i:INT;
END_VAR
FOR i:=1 TO g_mJntNum DO 
	IF m_jntOPMode[i]=DriverOPMode_PosTrq THEN
		// position controller and gravity feedforward
		m_cmdJntTrq[i]:=m_jntPIDCtrl[i].run(m_cmdJntPos[i],m_curJntPos[i],m_cmdJntVel[i],m_curJntVel[i]);
		m_cmdJntTrq[i]:=m_cmdJntTrq[i]+m_jntGravity[i];
		m_joints[i].updateCmds(DriverOPMode_Trq,m_cmdJntPos[i],m_cmdJntTrq[i]);
	ELSIF m_jntOPMode[i]=DriverOPMode_Trq THEN
		// gravity feedforward
		m_cmdJntTrq[i]:=m_cmdJntTrq[i]+m_jntGravity[i];
		m_cmdJntPos[i] :=m_curJntPos[i];
		m_joints[i].updateCmds(DriverOPMode_Trq,m_cmdJntPos[i],m_cmdJntTrq[i]);
	ELSE
		m_jntPIDCtrl[i].reset();
		m_cmdJntTrq[i]:=0;
	END_IF
	m_joints[i].updateCmds(m_jntOPMode[i],m_cmdJntPos[i],m_cmdJntTrq[i]);
END_FOR
END_METHOD

// update arm status, including kinematic and dynamic
METHOD PUBLIC updateStatus : BOOL
VAR_INPUT
END_VAR
VAR 
	i,j:INT;
END_VAR
// grip angle
m_gripAngle :=calcGripAngle();

// update joint data
FOR i:=1 TO g_mArmNum DO
	m_joints[i].updateStatus();
END_FOR

// get joint data
FOR i:=1 TO g_mJntNum DO
	m_curJntPos[i]:=m_joints[i].jntPos;
	m_curJntVel[i]:=m_joints[i].jntVel;
	m_curJntTrq[i]:=m_joints[i].jntTrq;
END_FOR 

// cartesion pose
forwardKinematic(m_curJntPos,m_curCartPose);

// jacobian
calcJaco(m_curJntPos,m_jaco);

// cartesian twist
m_curCartTwist:=Mat67Vec7(m_jaco,m_curJntVel);

// graivity compensation
m_gravityModel.run(m_curJntPos, m_jntGravity);
END_METHOD

END_FUNCTION_BLOCK

// ---- Robots/FB_Joint.TcPOU
FUNCTION_BLOCK FB_Joint
VAR_INPUT
END_VAR
VAR_OUTPUT
END_VAR
VAR
	// motor IO
	m_motorInputs AT%I*	:ST_MotorInputs;
	m_motorOutputs AT%Q* :ST_MotorOutputs;
	
	// device paramters
	m_incEncoderRes :DINT;
	m_absEncoderRes :DINT;
	m_motorReduction :LREAL;
	m_absEncoderReduction :LREAL;
	m_trqConst :LREAL;
	m_maxCurrent :LREAL;
	m_motorDir :INT;								
	m_asbEncoderDir :INT;
	m_minJntPos: LREAL;
	m_maxJntPos: LREAL;
	
	// convertion paramters
	m_trq2Current:LREAL;
	m_current2Trq:LREAL;
	
	// joint data
	m_curMotorPos :LREAL;
	m_curLinkPos :LREAL;
	m_curJntPos	:LREAL;
	m_curJntVel :LREAL;
	m_curJntTrq :	LREAL;
	m_cmdJntPos :LREAL;
	m_cmdJntVel :LREAL;
	m_cmdJntTrq :LREAL;
	m_lastJntPos :LREAL;
	
	// velocity filter
	m_jntVelLpf :FB_LowPassFilter;
	
	// command torque filter
	m_cmdTrqLpf :FB_LowPassFilter;
	
END_VAR

METHOD PUBLIC disable : BOOL
VAR_INPUT
END_VAR
m_motorOutputs.m_controlWord:=DriverCtrlWord_INIT;
disable:=true;
END_METHOD

METHOD PUBLIC enable : BOOL
VAR_INPUT
END_VAR
IF DriverStatusWord_INIT = m_motorInputs.m_statusWord THEN
	m_motorOutputs.m_controlWord:=DriverCtrlWord_PREOP;
	enable := FALSE;
ELSIF DriverStatusWord_PREOP = m_motorInputs.m_statusWord THEN
	m_motorOutputs.m_controlWord:=DriverCtrlWord_OP;
	enable :=  FALSE;
ELSIF DriverStatusWord_OP = m_motorInputs.m_statusWord THEN
	enable :=  TRUE;
ELSE
	m_motorOutputs.m_controlWord:=DriverCtrlWord_INIT;
	enable :=  FALSE;
END_IF
END_METHOD

METHOD PROTECTED encoder2Pos : BOOL
VAR_INPUT
END_VAR
//m_curMotorPos:=
//m_curLinkPos:=

// use motor pos as joint pos
m_curJntPos:=m_curMotorPos;
END_METHOD

METHOD PUBLIC init : BOOL
VAR_INPUT
	i_armIdx :INT;
	i_jntIdx :INT;
END_VAR
// hardware parameters
m_incEncoderRes :=g_incEncoderRes[i_jntIdx];
m_absEncoderRes :=g_absEncoderRes[i_jntIdx];
m_motorReduction :=g_motorReduction[i_jntIdx];
m_absEncoderReduction :=g_absEncoderReduction[i_jntIdx];
m_trqConst :=g_motorTrqConst[i_jntIdx];
m_maxCurrent :=g_motorMaxCurrent[i_jntIdx];
m_motorDir :=g_motorDir[i_armIdx,i_jntIdx];								
m_asbEncoderDir :=g_asbEncoderDir[i_armIdx,i_jntIdx];
m_minJntPos	:=g_minJntPos[i_armIdx,i_jntIdx];
m_maxJntPos	:=g_maxJntPos[i_armIdx,i_jntIdx];

m_trq2Current:=m_motorDir * 1000.0/(m_trqConst*m_motorReduction);
m_current2Trq:=m_motorDir * (m_trqConst*m_motorReduction)/1000.0;

// motor data init
encoder2Pos();
m_curJntVel:=0;
m_curJntTrq :=0;
m_cmdJntPos :=m_curJntPos;
m_cmdJntVel :=0.0;
m_cmdJntTrq :=0.0;
m_lastJntPos :=m_curJntPos;
m_jntVelLpf.init(1, g_curJntVelLpfCutoffFreq, g_armControlFreq);
m_cmdTrqLpf.init(1, g_cmdJntTrqLpfCutoffFreq, g_armControlFreq);

// driver init value
m_motorOutputs.m_controlWord:=DriverCtrlWord_INIT;
m_motorOutputs.m_controlWord:=DriverOPMode_Pos;
m_motorOutputs.m_cmdCurrent:=0;
m_motorOutputs.m_cmdMotorEncoder:=m_motorInputs.m_motorEncoder;
END_METHOD

PROPERTY jntPos : LREAL
GET
jntPos := m_curJntPos;
END_GET
END_PROPERTY

PROPERTY jntTrq : LREAL
GET
jntTrq:=m_curJntTrq;
END_GET
END_PROPERTY

PROPERTY jntVel : LREAL
GET
jntVel := m_curJntVel;
END_GET
END_PROPERTY

PROPERTY PUBLIC linkPos : LREAL
GET
linkPos:=m_curLinkPos;
END_GET
END_PROPERTY

PROPERTY PUBLIC motorPos : LREAL
GET
motorPos := m_curMotorPos;
END_GET
END_PROPERTY

// TODO
METHOD PROTECTED pos2Encoder : DINT
VAR_INPUT
	i_jntPos :LREAL;
END_VAR

VAR
END_VAR
//m_motorOutputs.m_cmdMotorEncoder:=
END_METHOD

METHOD PUBLIC updateCmds : BOOL
VAR_INPUT
	i_opMode : E_DriverOPMode;
	i_cmdPos :LREAL;
	i_cmdTrq :LREAL;
END_VAR
m_motorOutputs.m_opMode:=INT_TO_SINT( i_opMode);
// pos mode
IF i_opMode = DriverOPMode_Pos THEN
	m_motorOutputs.m_cmdCurrent:=0;
	m_motorOutputs.m_cmdMotorEncoder :=pos2Encoder(i_cmdPos);
ELSIF i_opMode = DriverOPMode_Trq THEN
	m_motorOutputs.m_cmdCurrent:=LREAL_TO_DINT(i_cmdTrq*m_trq2Current);
	m_motorOutputs.m_cmdMotorEncoder :=m_motorInputs.m_motorEncoder; 
END_IF
END_METHOD

METHOD PUBLIC updateStatus : BOOL
VAR_INPUT
END_VAR
// get joint position
encoder2Pos();

// compute joint velocity
m_curJntVel:= (m_curJntPos-m_lastJntPos)/g_armControlLoopInterval;
m_curJntVel := m_jntVelLpf.run(m_curJntVel);

m_curJntTrq := m_motorInputs.m_current * m_current2Trq;
END_METHOD

END_FUNCTION_BLOCK

// ---- FBs_dynamics/FB_MasterGravity.TcPOU
FUNCTION_BLOCK FB_MasterGravity
VAR_INPUT
END_VAR
VAR_OUTPUT
END_VAR
VAR
	// arm index
	m_armIdx :INT;
	
	(*graParam=[ 2.7244*m3 + 2.7244*m4 + 2.7244*m5 + 2.7244*m6 + 9.8*mx2 + 9.8*mx9,
            	9.8*my2 + 9.8*my9,
			 	3.577*m4 + 3.577*m5 + 3.577*m6 + 0.49*m9 + 9.8*mx3 + 9.8*mx8
           		1.5827*m4 + 1.5827*m5 + 1.5827*m6 + 9.8*my3 + 9.8*my8 + 9.8*mz4
            	mz5-my4,	my5+mz6,  	mx4,   	mx5, 	mx6,   	my6
            	preF2,   k2,   preF3,    k3,    preF5   k5]*)
	m_gravityParam :ARRAY[1..16] OF REAL;
	// spring2 [L0, b1, b2, l1, r0]
	m_spring2Param :ARRAY[1..5] OF LREAL;
	// spring3 [L0, b1, b2, l1, r0,d]
	m_spring3Param :ARRAY[1..6] OF LREAL;
	// spring5 [L0, s1, L1, r0, beta]
	m_spring5Param :ARRAY[1..5] OF LREAL;
END_VAR

METHOD protected getRegMat : BOOL
VAR_INPUT
	// 0 for left, 1 for right
	i_armIdx:INT;
END_VAR
VAR_IN_OUT CONSTANT
	// position of all the active joint
	i_jointPos:ARRAY[1..7] OF LREAL;
END_VAR
VAR_IN_OUT
	o_regMat:ARRAY[1..5,1..16] OF LREAL;
END_VAR
VAR
	q2,q8,q4,q5,q6:LREAL;
	i,j :INT;
END_VAR
q2:=i_jointPos[2];
q8:=i_jointPos[3];
q4:=i_jointPos[4];
q5:=i_jointPos[5];
q6:=i_jointPos[6];

FOR i:=1 TO 5 DO
	FOR j:=1 TO 16 DO
		o_regMat[i,j]:=0;
	END_FOR
END_FOR

// active joint 2
o_regMat[1,1]:=COS(q2);
o_regMat[1,2]:=-SIN(q2); 
o_regMat[1,3] := 0;
o_regMat[1,4] :=   0;
o_regMat[1,5] := - 4.9*(COS(q2 - q4) - COS(q4 - q2 + 2.0*q8));
o_regMat[1,6] :=  9.8*COS(q4 - q2 + q8)*SIN(q5)*SIN(q8);
o_regMat[1,7] :=   - 4.9*(SIN(q2 - q4) + SIN(q4 - q2 + 2.0*q8));
o_regMat[1,8] :=   - 9.8*COS(q4 - q2 + q8)*COS(q5)*SIN(q8);
o_regMat[1,9] :=  9.8*SIN(q8)*(SIN(q4 - q2 + q8)*SIN(q6) - COS(q4 - q2 + q8)*COS(q5)*COS(q6));
o_regMat[1,10] :=9.8*SIN(q8)*(SIN(q4 - q2 + q8)*COS(q6) + COS(q4 - q2 + q8)*COS(q5)*SIN(q6));
spring2RegMat(q2, o_preF=>o_regMat[1,11], o_stiff=>o_regMat[1,12]);
o_regMat[1,11]:=-o_regMat[1,11];         
o_regMat[1,12]:=-o_regMat[1,12];

// active joint3
o_regMat[2,3]:= COS(q8);
o_regMat[2,4]:= - SIN(q8);
o_regMat[2,5]:= -9.8*(COS(2.0*q8)*COS(q2)*COS(q4) + COS(2.0*q8)*SIN(q2)*SIN(q4) - SIN(2.0*q8)*COS(q2)*SIN(q4) + SIN(2.0*q8)*COS(q4)*SIN(q2));
o_regMat[2,6]:= -9.8*(COS(q5)*SIN(q8) + COS(2.0*q8)*COS(q2)*SIN(q4)*SIN(q5) - COS(2.0*q8)*COS(q4)*SIN(q2)*SIN(q5) + SIN(2.0*q8)*COS(q2)*COS(q4)*SIN(q5) + SIN(2.0*q8)*SIN(q2)*SIN(q4)*SIN(q5));
o_regMat[2,7]:= 9.8*(COS(2.0*q8)*COS(q2)*SIN(q4) - COS(2.0*q8)*COS(q4)*SIN(q2) + SIN(2.0*q8)*COS(q2)*COS(q4) + SIN(2.0*q8)*SIN(q2)*SIN(q4));
o_regMat[2,8]:= 9.8*(COS(2.0*q8)*COS(q2)*COS(q5)*SIN(q4) - SIN(q5)*SIN(q8) - COS(2.0*q8)*COS(q4)*COS(q5)*SIN(q2) + SIN(2.0*q8)*COS(q2)*COS(q4)*COS(q5) + SIN(2.0*q8)*COS(q5)*SIN(q2)*SIN(q4));
o_regMat[2,9]:= 9.8*(COS(2.0*q8)*COS(q2)*COS(q4)*SIN(q6) - COS(q6)*SIN(q5)*SIN(q8) + COS(2.0*q8)*SIN(q2)*SIN(q4)*SIN(q6) - SIN(2.0*q8)*COS(q2)*SIN(q4)*SIN(q6) + SIN(2.0*q8)*COS(q4)*SIN(q2)*SIN(q6) + COS(2.0*q8)*COS(q2)*COS(q5)*COS(q6)*SIN(q4) - COS(2.0*q8)*COS(q4)*COS(q5)*COS(q6)*SIN(q2) + SIN(2.0*q8)*COS(q2)*COS(q4)*COS(q5)*COS(q6) + SIN(2.0*q8)*COS(q5)*COS(q6)*SIN(q2)*SIN(q4)); 
o_regMat[2,10]:= 9.8*(SIN(q5)*SIN(q6)*SIN(q8) + COS(2.0*q8)*COS(q2)*COS(q4)*COS(q6) + COS(2.0*q8)*COS(q6)*SIN(q2)*SIN(q4) - SIN(2.0*q8)*COS(q2)*COS(q6)*SIN(q4) + SIN(2.0*q8)*COS(q4)*COS(q6)*SIN(q2) - COS(2.0*q8)*COS(q2)*COS(q5)*SIN(q4)*SIN(q6) + COS(2.0*q8)*COS(q4)*COS(q5)*SIN(q2)*SIN(q6) - SIN(2.0*q8)*COS(q2)*COS(q4)*COS(q5)*SIN(q6) - SIN(2.0*q8)*COS(q5)*SIN(q2)*SIN(q4)*SIN(q6));
spring3RegMat(q8, o_preF=>o_regMat[2,13], o_stiff=>o_regMat[2,14]);
o_regMat[2,13]:=-o_regMat[2,13];
o_regMat[2,14]:=-o_regMat[2,14];

// active joint4
o_regMat[3,5]:= 9.8*SIN(q4 - q2 + q8)*SIN(q8);
o_regMat[3,6]:= - 9.8*COS(q4 - q2 + q8)*SIN(q5)*SIN(q8);
o_regMat[3,7]:= 9.8*COS(q4 - q2 + q8)*SIN(q8);
o_regMat[3,8]:= 9.8*COS(q4 - q2 + q8)*COS(q5)*SIN(q8);
o_regMat[3,9]:= - 9.8 *SIN(q8)*(SIN(q4 - q2 + q8)*SIN(q6) - COS(q4 - q2 + q8)*COS(q5)*COS(q6));
o_regMat[3,10]:= - 9.8*SIN(q8)*(SIN(q4 - q2 + q8)*COS(q6) + COS(q4 - q2 + q8)*COS(q5)*SIN(q6));
              
// active joint5
o_regMat[4,6]:= -9.8* (COS(q8)*SIN(q5) + SIN(q4 - q2 + q8)*COS(q5)*SIN(q8));
o_regMat[4,7]:= 0;
o_regMat[4,8]:= 9.8* (COS(q5)*COS(q8) - SIN(q4 - q2 + q8)*SIN(q5)*SIN(q8));
o_regMat[4,9]:= 9.8*COS(q6)*(COS(q5)*COS(q8) - SIN(q4 - q2 + q8)*SIN(q5)*SIN(q8));
o_regMat[4,10]:= -9.8*SIN(q6)*(COS(q5)*COS(q8) - SIN(q4 - q2 + q8)*SIN(q5)*SIN(q8));
spring5RegMat(q5,i_armIdx, o_preF=>o_regMat[4,15], o_stiff=>o_regMat[4,16]);
o_regMat[4,15]:=-o_regMat[4,15];
o_regMat[4,16]:=-o_regMat[4,16];

// active joint5
o_regMat[5,9]:= -9.8*(COS(q8)*SIN(q5)*SIN(q6) - COS(q4 - q2 + q8)*COS(q6)*SIN(q8) + SIN(q4 - q2 + q8)*COS(q5)*SIN(q6)*SIN(q8));
o_regMat[5,10]:= -9.8*(COS(q4 - q2 + q8)*SIN(q6)*SIN(q8) + COS(q6)*COS(q8)*SIN(q5) + SIN(q4 - q2 + q8)*COS(q5)*COS(q6)*SIN(q8));
END_METHOD

METHOD PUBLIC init : BOOL
VAR_INPUT
	i_armIdx :INT;
END_VAR
VAR
	i:INT;
END_VAR
m_armIdx:=i_armIdx;

FOR i:=1 TO 16 DO
	m_gravityParam[i]:=g_gravityParam[m_armIdx, i];
END_FOR

FOR i:=1 TO 5 DO
	m_spring2Param[i]:=g_spring2Param[i];
	m_spring3Param[i]:=g_spring3Param[i];
	m_spring5Param[i]:=g_spring5Param[i];
END_FOR
m_spring3Param[6]:=g_spring3Param[6];
END_METHOD

METHOD PUBLIC run : BOOL
VAR_IN_OUT CONSTANT
	// active joint position
	i_jntPos :vec7d;
END_VAR
VAR_IN_OUT
	r_gravity :Vec7d;
END_VAR
VAR

	// position of all the active joint
	m_leftJntPos:ARRAY[1..7] OF LREAL;
	m_rightJntPos:ARRAY[1..7] OF LREAL;
	
	// gravity regression matrix
	regMat:ARRAY[1..5,1..16] OF LREAL;
	
	i,j:INT;
END_VAR
getRegMat(m_armIdx,i_jntPos,regMat);

FOR i:=2 TO 6 DO
	FOR j:=1 TO 16 DO
		r_gravity[i]:=r_gravity[i]+regMat[i-1,j]*m_gravityParam[j];
	END_FOR
END_FOR
END_METHOD

(*spring force F = preF+k(L-L0)
% torque trq=F*t=preF*t+k*t*(L-L0)=[t, t*(L-L0)]*[preF,k]'
% this function return [t, t(L-L0)]*)
METHOD PROTECTED spring2RegMat : BOOL
VAR_INPUT
	i_q2:LREAL;
END_VAR

VAR
	// spring paramters
	L0, b1, b2, l1, r0 : LREAL;

	theta,length,t:LREAL;  
	
END_VAR

VAR_OUTPUT
	o_preF:LREAL;
	o_stiff:LREAL;
END_VAR
L0:=m_spring2Param[1]; 
b1:=m_spring2Param[2]; 
b2:=m_spring2Param[3]; 
l1:=m_spring2Param[4]; 
r0:=m_spring2Param[5]; 

L0:=L0+b1+b2;
 
//spring length
theta:=i_q2+90*g_deg2Rad;
length:=SQRT(l1*l1+r0*r0+2*l1*r0*COS(theta));

//force arm
t:=r0*l1*SIN(theta)/Length;

//torque direction is determined by theta(or t)
o_preF:=t;
o_stiff:=t*(length-L0);
END_METHOD

(*spring force F = preF+k(L-L0)
% torque trq=F*t=preF*t+k*t*(L-L0)=[t, t*(L-L0)]*[preF,k]'
% this function return [t, t(L-L0)]*)
METHOD PROTECTED spring3RegMat : BOOL
VAR_INPUT
	i_q3:LREAL;
END_VAR

VAR
	// spring paramters
	L0, b1, b2, l1, r0, d: LREAL;

	alpha, beta,tanBeta, length,t:LREAL;  
	
	spring: INT;
END_VAR

VAR_OUTPUT
	o_preF:LREAL;
	o_stiff:LREAL;
END_VAR
L0:=m_spring3Param[1]; 
b1:=m_spring3Param[2]; 
b2:=m_spring3Param[3]; 
l1:=m_spring3Param[4]; 
r0:=m_spring3Param[5];
d:=m_spring3Param[6];

L0:=L0+b1+b2;
 
// spring length
    alpha:=i_q3+90*g_deg2Rad;
    tanBeta:=(r0*SIN(alpha)+d)/(l1+r0*COS(alpha));
    beta:=ATAN(tanBeta);
    length:=d/SIN(beta)+r0*SIN(alpha)/SIN(beta);
    
// force arm
    t:=(l1-d*cot(beta))*SIN(beta);
    
// torque direction is determined by theta(or t)
    o_preF:=t;
    o_stiff:=t*(length-L0);
END_METHOD

(*spring force F = preF+k(L-L0)
 torque trq=F*t=preF*t+k*t*(L-L0)=[t, t*(L-L0)]*[preF,k]'
 this function return [t, t(L-L0)]
 armIdx, 0 for left arm , 1 for right arm]*)
METHOD PROTECTED spring5RegMat : BOOL
VAR_INPUT
	i_q5:LREAL;
	i_armIdx:INT;
END_VAR

VAR
	// spring paramters
	L0, s1, L1, r0, beta: LREAL;

	theta, length,t:LREAL;  
	
	spring: INT;
	joint: INT;
	armIdx: INT;
	b1: LREAL;
END_VAR

VAR_OUTPUT
	o_preF:LREAL;
	o_stiff:LREAL;
END_VAR
L0:=m_spring5Param[1]; 
s1:=m_spring5Param[2]; 
L1:=m_spring5Param[3]; 
r0:=m_spring5Param[4]; 
beta:=m_spring5Param[5];

L0:=L0+s1;
 
// joint 5 motion angle
IF i_armIdx=0 THEN 
	theta:=i_q5-pi;// left arm
ELSIF i_armIdx=1 THEN 
	theta:=pi-i_q5; // right arm
END_IF

// spring length and force arm
length:=SQRT(L1*L1+r0*r0+2*L1*r0*COS(theta+beta));
t:=L1*r0*SIN(theta+beta)/length;

// torque direction is determined by t
IF i_armIdx = 0 THEN 
	o_preF:=t;
	o_stiff:=t*(length-L0);
else
	o_preF:=-t;
	o_stiff:=-t*(length-L0);
END_IF
END_METHOD

END_FUNCTION_BLOCK

// ---- Maths/cot.TcPOU
FUNCTION cot : lreal
VAR_INPUT
	i_angle:LREAL;
END_VAR
VAR
END_VAR

cot:=COS(i_angle)/SIN(i_angle);

END_FUNCTION

// ---- Maths/mat67Vec7.TcPOU
FUNCTION mat67Vec7 : Vec6d
VAR_IN_OUT CONSTANT
	i_mat :ARRAY[1..6,1..7] OF LREAL;
	i_vec :ARRAY[1..7] OF LREAL;
END_VAR
VAR
	i,j : INT ;
END_VAR

FOR i:=1 TO 6 DO
	Mat67Vec7[i]:=0.0;
	FOR j:=1 TO 7 DO
		Mat67Vec7[i]:=Mat67Vec7[i]+i_mat[i,j]*i_vec[j];
	END_FOR
END_FOR

END_FUNCTION

// ---- FBs_Controller/FBRedunOriControl.TcPOU
// Author: Feijian Ni
// Date: 2023.11.22
FUNCTION_BLOCK FBRedunOriControl
VAR_INPUT
END_VAR
VAR_OUTPUT
END_VAR
VAR
	//TODO: move to GVLs 
	// control paramters for redundant joint4 position control
	m_redunJntKp: LREAL:=1;
	m_redunJntKd:LREAL:=0.1;
	m_redunJntKi:LREAL:=1;
	m_redunJntKiLimit: LREAL:=500;
	m_redunJntCtrlLimit:LREAL:=1000;
	m_jntTargetPosLpfCutoffFreq:LREAL:=10;
	m_curJntVelLpfCutoffFreq:LREAL:=30;

	// max command joint velocity
	m_maxJntVel:LREAL:= deg2rad(30);
	
	// filter for target joint position
	m_cmdPosLpf:ARRAY[1..2] OF FB_LowPassFilter;
	
	// final target position of joint4 in motor (not DH , same for blow defination) 
	m_targetJntPos:ARRAY[1..2] OF LREAL;
	
	// position tracking error
	m_posErr:ARRAY[1..2] OF LREAL;
	
	// command joint4 position and veloicty in motor for next cycle
	m_cmdJntPos:ARRAY[1..2] OF LREAL;
	m_cmdJntVel:ARRAY[1..2] OF LREAL;

	// current joint4 position and veloicty in motor
	m_curJntPos:ARRAY[1..2] OF LREAL;
	m_curJntVel:ARRAY[1..2] OF LREAL;
	
	// last joint4 position in motor
	m_lastJntPos:ARRAY[1..2] OF LREAL;
	
	// filter for current joint velocity
	m_curJntVelLpf:ARRAY[1..2] OF FB_LowPassFilter;
	
	// PID for joint position
	m_jntPIDCtrl:ARRAY[1..2] OF FB_PID;
	m_jntCtrlTrq:ARRAY[1..2] OF LREAL;
	
	// orientation joints control torque in redundance sapce
	m_redunCtrlTrq:ARRAY[1..2,1..4] OF LREAL;
	
	// master jacobian solver
	m_jacobianSolver:Robot_Jacobian_matrix_C0;
	posOriJaco:ARRAY[1..6,1..7] OF LREAL;
	Jt:ARRAY[1..7,1..6] OF LREAL;
	JJt:ARRAY[1..6,1..6] OF LREAL;
	invJJt:ARRAY[1..6,1..6] OF LREAL;
	pinvJt:ARRAY[1..6,1..7] OF LREAL;
	JtPinvJt:ARRAY[1..7,1..7] OF LREAL;
	nullSpacePinvJt:ARRAY[1..7,1..7] OF LREAL;
	
END_VAR

METHOD PROTECTED DH2MotorPos : BOOL
VAR_INPUT
	// target joint4 DH position
	i_targetDHPos:ARRAY[1..2] OF LREAL;
	
	// current joint4 DH position
	i_currentDHPos:ARRAY[1..2] OF LREAL;
END_VAR

VAR_OUTPUT
	// target joint4 motor position
	o_targetMotorPos:ARRAY[1..2] OF LREAL;
	
	// current joint4 motor position
	o_currentMotorPos:ARRAY[1..2] OF LREAL;
END_VAR

VAR
	// active joint3 position
	q2,q3,q4,q8:LREAL;
	
END_VAR
// left arm
q2:=Robot_Status.robot_current_joint_position_v2[1,2];
q3:=Robot_Status.robot_current_joint_position_v2[1,3];
q4:=Robot_Status.robot_current_joint_position_v2[1,4];
// q8 = q3+q2;
q8:=q3+q2;
// q4Jnt= q4motor+q8-q2-90;
o_targetMotorPos[1]:=i_targetDHPos[1]-q8+q2+deg2rad(90);
o_currentMotorPos[1]:=i_currentDHPos[1]-q8+q2+deg2rad(90);

// right arm
q2:=Robot_Status.robot_current_joint_position_v2[2,2];
q3:=Robot_Status.robot_current_joint_position_v2[2,3];
q4:=Robot_Status.robot_current_joint_position_v2[2,4];
// q8 = q3+q2;
q8:=q3+q2;
// q4Jnt= q4motor+q8-q2-90;
o_targetMotorPos[2]:=i_targetDHPos[2]-q8+q2+deg2rad(90);
o_currentMotorPos[2]:=i_currentDHPos[2]-q8+q2+deg2rad(90);
END_METHOD

METHOD init : BOOL
VAR
	i,j:INT;
	currentRatioMotor2Jnt:LREAL;
END_VAR
// reset joint position 
m_curJntPos[1]:=Robot_Status.robot_current_joint_position_v2[1,4];
m_curJntPos[2]:=Robot_Status.robot_current_joint_position_v2[2,4];
m_targetJntPos:=m_curJntPos;
DH2MotorPos(m_targetJntPos,m_curJntPos, o_targetMotorPos=>m_targetJntPos,o_currentMotorPos=>m_curJntPos);
m_cmdJntPos:=m_curJntPos;
m_lastJntPos:=m_curJntPos;

FOR i:=1 TO 2  DO 
	// init velocity
	m_cmdJntVel[i]:=0;
	m_curJntVel[i]:=0;
	m_posErr[i]:=0;
	
	// init controller
	currentRatioMotor2Jnt:=GVL_system_parameters.transmition_efficiency[i,4]*GVL_system_parameters.torque_constant[i,4]
							*GVL_system_parameters.transmission_ratio[i, 4]/1000;
	m_jntPIDCtrl[i].init(GVL_system_parameters.cycle_robot,m_redunJntKp,m_redunJntKd,m_redunJntKi,
		m_redunJntKiLimit* currentRatioMotor2Jnt,	m_redunJntCtrlLimit*currentRatioMotor2Jnt);
	
	// init filter
	m_cmdPosLpf[i].init(i_filterOrd:=1,i_cutoffFreq:=m_jntTargetPosLpfCutoffFreq,i_sampleFreq:=1000);
	m_curJntVelLpf[i].init(i_filterOrd:=1,i_cutoffFreq:=m_curJntVelLpfCutoffFreq,i_sampleFreq:=1000);
END_FOR
END_METHOD

METHOD run : BOOL
VAR_INPUT
	// target position for left and right joint4
	i_targetJntPos:ARRAY[1..2] OF LREAL;

END_VAR

VAR_OUTPUT
	// control torque for last four orientation joints
	o_cmdCtrlTrq:ARRAY[1..2, 1..4] OF LREAL :=[8(0.0)];
END_VAR

VAR
	i,j,k: INT;
	currentDHPos:ARRAY[1..2] OF LREAL;
	jacoTransCalc : Jacobian_Matrix_Tr;
	matrixInvCalc: matrix_fun_inv;
	invFlag:BOOL;
	scale:LREAL;
END_VAR
// convert target and current joint position from DH to motor
currentDHPos[1]:=Robot_Status.robot_current_joint_position_v2[1,4];
currentDHPos[2]:=Robot_Status.robot_current_joint_position_v2[2,4];
DH2MotorPos(i_targetJntPos,currentDHPos,o_targetMotorPos=>m_targetJntPos, o_currentMotorPos=>m_curJntPos);

FOR i:=1 TO 2 DO
	// fitl target joint position
	m_targetJntPos[i]:=m_cmdPosLpf[i].run(m_targetJntPos[i]);

	// get current joint velocity
	m_curJntVel[i]:=(m_curJntPos[i]-m_lastJntPos[i])/GVL_system_parameters.cycle_robot;
	m_curJntVel[i]:=m_curJntVelLpf[i].run(m_curJntVel[i]);
	m_lastJntPos[i]:=m_curJntPos[i];

	// interpolate command position
	m_cmdJntVel[i]:=LIMIT(-m_maxJntVel,(m_targetJntPos[i]-m_cmdJntPos[i])/GVL_system_parameters.cycle_robot, m_maxJntVel);
	m_cmdJntPos[i]:=m_cmdJntPos[i]+m_cmdJntVel[i]*GVL_system_parameters.cycle_robot;

	// joint position control torque control
	m_posErr[i]:=m_cmdJntPos[i]-m_curJntPos[i];
	m_jntCtrlTrq[i]:=m_jntPIDCtrl[i].run(m_cmdJntPos[i],m_curJntPos[i], m_cmdJntVel[i], m_curJntVel[i]);
END_FOR

// control current
o_cmdCtrlTrq[1,1]:=m_jntCtrlTrq[1];
o_cmdCtrlTrq[2,1]:=m_jntCtrlTrq[2];

// project control torque to nullspace
m_jacobianSolver(arm_id:= 1, current_Joint_position:= Robot_Status.Robot_current_Joint_position[1], Jacobian_matrix_0=> posOriJaco);
jacoTransCalc(Jacobian_matrix:=posOriJaco,Jacobian_matrix_tr=>Jt);
// J*Jt
FOR i:=1 TO 6 DO
	FOR j:=1 TO 6 DO
		JJt[i,j]:=0;
		FOR k:=1 TO 7 DO
			JJt[i,j]:=JJt[i,j]+posOriJaco[i,k]*Jt[k,j];
		END_FOR
	END_FOR
END_FOR

// inv(JJt)
matrixInvCalc(input_matrix:=JJt,output_matrix=>invJJt, succeed=>invFlag);
IF invFlag=FALSE THEN
	run:=FALSE;
	RETURN;
END_IF

// pinv(Jt)=inv(JJt)*J
FOR i:=1 TO 6 DO
	FOR j:=1 TO 7 DO
		pinvJt[i,j]:=0;
		FOR k:=1 TO 6 DO
			pinvJt[i,j]:=pinvJt[i,j]+invJJt[i,k]*posOriJaco[k,j];
		END_FOR
	END_FOR
END_FOR

// Jt*Pinv(Jt)
FOR i:=1 TO 7 DO
	FOR j:=1 TO 7 DO
		JtPinvJt[i,j]:=0;
		FOR k:=1 TO 6 DO
			JtPinvJt[i,j]:=JtPinvJt[i,j]+Jt[i,k]*pinvJt[k,j];
		END_FOR
	END_FOR
END_FOR
 
// nullspace of pinv(Jt): I-Jt*Pinv(Jt)
FOR i:=1 TO 7 DO
	FOR j:=1 TO 7 DO
		IF i = j THEN
			nullSpacePinvJt[i,j]:=1-JtPinvJt[i,j];
		ELSE
			nullSpacePinvJt[i,j]:=-JtPinvJt[i,j];
		END_IF
	END_FOR
END_FOR

IF ABS(nullSpacePinvJt[4,4])>0.001 THEN 
	scale :=1/nullSpacePinvJt[4,4];
	o_cmdCtrlTrq[1,2]:=scale*nullSpacePinvJt[5,4]*o_cmdCtrlTrq[1,1];
	o_cmdCtrlTrq[1,3]:=scale*nullSpacePinvJt[6,4]*o_cmdCtrlTrq[1,1];
	o_cmdCtrlTrq[1,4]:=scale*nullSpacePinvJt[7,4]*o_cmdCtrlTrq[1,1];
ELSE
	o_cmdCtrlTrq[1,2]:=0;
	o_cmdCtrlTrq[1,3]:=0;
	o_cmdCtrlTrq[1,4]:=0;
END_IF
END_METHOD

END_FUNCTION_BLOCK

// ---- MAIN.TcPOU
PROGRAM MAIN
VAR
	// flag to init robot
	g_robotInit :BOOL :=FALSE;
	
	// master robot
	g_masterRobot:FB_MasterRobot;
	
	// master robot information, export to other task or device
	m_masterStatus AT %Q* :ST_MasterStatus;
	
	// cart information, import from other task
	m_cartStatus AT %I*:ST_CartStatus;
	
	// slave robot information, import from other device
	m_slaveStatus AT %I*:ST_SlaveStatus;
	
END_VAR



IF g_robotInit =FALSE THEN
	g_masterRobot.Init();
	g_robotInit:=TRUE;
END_IF

g_masterRobot.run(m_cartStatus,m_slaveStatus);

END_PROGRAM

// ---- Robots/FB_MasterRobot.TcPOU
FUNCTION_BLOCK FB_MasterRobot
VAR_INPUT
END_VAR
VAR_OUTPUT
END_VAR
VAR
	// arm shoulders frame in monitor
	m_shoulderPose :ARRAY[1..2] OF ST_Frame;
	
	// master arms, responsible for arm kinematic and control
	m_masterArms :ARRAY[1..2] OF FB_MasterArm;
	
	// current and las arm state
	m_masterArmState:ARRAY[1..2] OF E_masterArmState:=[E_masterArmState.MasterArmState_Init,E_masterArmState.MasterArmState_Init];
	m_lastMasterArmState:ARRAY[1..2] OF E_masterArmState:=[E_masterArmState.MasterArmState_Init,E_masterArmState.MasterArmState_Init];
	
	// index(1 to 4) of slave arm which is tele-linked to master arm
	m_slaveArmIdx:ARRAY[1..2] OF E_MatchedSlaveArmIdx:=[MatchedSlaveArmIdx_NULL, MatchedSlaveArmIdx_null];
	
	// arm controller
	m_armCtrl :I_MasterArmCtrl;
END_VAR

METHOD PUBLIC Init : BOOL
VAR_INPUT
END_VAR
VAR
	i:INT;
END_VAR
FOR i:=1 TO g_mArmNum DO
	m_masterArms[i].Init(i);
	m_masterArmState[i]:=MasterArmState_Init;
	m_lastMasterArmState[i]:=MasterArmState_Init;
	m_slaveArmIdx[i]:=MatchedSlaveArmIdx_NULL;
END_FOR

m_shoulderPose[1].m_pos[1]:= g_armShoulderDistance/2.0;
m_shoulderPose[2].m_pos[1]:= -g_armShoulderDistance/2.0;
END_METHOD

METHOD PUBLIC run : BOOL
VAR_IN_OUT CONSTANT
	i_cartStatus :ST_CartStatus;
	
	i_slaveStatus :ST_SlaveStatus;
END_VAR
VAR
	i:INT;
END_VAR
// state machine transition
stateMachine(i_cartStatus,i_slaveStatus);

// update shoulder pose (wrt monitor)
m_shoulderPose[1].m_rot:=rotY(m_shoulderPose[1].m_rot,i_cartStatus.m_monitorAngle);
m_shoulderPose[2].m_rot:=rotY(m_shoulderPose[2].m_rot,i_cartStatus.m_monitorAngle);

// update master arm kinematics
FOR i:=1 TO g_mArmNum DO
	m_masterArms[i].updateStatus();
END_FOR

// run controller
m_armCtrl.run(m_shoulderPose,i_slaveStatus, m_masterArms);

// update commands to drivers
FOR i:=1 TO g_mArmNum DO
	m_masterArms[i].updateCmds();
END_FOR
END_METHOD

// state machine check and transit 
METHOD PROTECTED stateMachine : BOOL
VAR_IN_OUT CONSTANT
	i_cartStatus :ST_CartStatus;
	
	i_slaveStatus :ST_SlaveStatus;
END_VAR
END_METHOD

END_FUNCTION_BLOCK

// ---- Maths/addVec3.TcPOU
FUNCTION addVec3 : vec3d
VAR_IN_OUT CONSTANT
	i_vec1 :Mat3d;
	i_vec2 :Mat3d;
END_VAR
VAR
	i: INT ;
END_VAR

FOR i:=1 TO 3 DO 
	addVec3[i]:=i_vec1[i]+i_vec2[i];
END_FOR

END_FUNCTION

// ---- Maths/mat3Vec3.TcPOU
FUNCTION mat3Vec3 : vec3d
VAR_IN_OUT CONSTANT
	i_mat :Mat3d;
	i_vec :Vec3d;
END_VAR
VAR
	i,j : INT ;
END_VAR

FOR i:=1 TO 3 DO
	mat3Vec3[i]:=0.0;
	FOR j:=1 TO 3 DO
		mat3Vec3[i]:=mat3Vec3[i]+i_mat[i,j]*i_vec[j];
	END_FOR
END_FOR

END_FUNCTION

// ---- Maths/rotZ.TcPOU
FUNCTION rotZ : mat3d
VAR_IN_OUT CONSTANT
	i_mat : Mat3d;
	i_ang : LREAL;
END_VAR
VAR
	rot :Mat3d := g_eye3d;
END_VAR

rot[1,1]:=COS(i_ang);
rot[2,2]:=rot[1,1];
rot[2,1]:=SIN(i_ang);
rot[1,2]:=-rot[2,1];
rotZ := mat3Mat3(i_mat, rot);

END_FUNCTION

// ---- Maths/rotX.TcPOU
FUNCTION rotX : mat3d
VAR_IN_OUT CONSTANT
	i_mat : Mat3d;
	i_ang : LREAL;
END_VAR
VAR
	rot :Mat3d := g_eye3d;
END_VAR

rot[2,2]:=COS(i_ang);
rot[3,3]:=rot[2,2];
rot[3,2]:=SIN(i_ang);
rot[2,3]:=-rot[3,2];
rotX := mat3Mat3(i_mat, rot);

END_FUNCTION

// ---- Maths/transform.TcPOU
FUNCTION transform : ST_Frame
VAR_IN_OUT CONSTANT
	i_frame1 :ST_Frame;
	i_frame2 :ST_Frame;
END_VAR
VAR
END_VAR

transform.m_rot := mat3Mat3(i_frame1.m_rot, i_frame2.m_rot);
transform.m_pos := mat3Vec3(i_frame1.m_rot, i_frame2.m_pos);
transform.m_pos :=addVec3(transform.m_pos,i_frame1.m_pos);

END_FUNCTION
